{attribute 'GeneratedUsingTerminal: IODEVICETYPE_ETHERCATPROT'}
{attribute addProperty BoxType "IODEVICETYPE_ETHERCATPROT"}
{attribute addProperty Id "DevCtrlAT %Q*UINT2Frm0CtrlAT %Q*UINT2Frm0WcCtrlAT %Q*UINT2Frm1CtrlAT %Q*UINT2Frm1WcCtrlAT %Q*UINT2Frm2CtrlAT %Q*UINT2Frm2WcCtrlAT %Q*UINT2Frm3CtrlAT %Q*UINT2Frm3WcCtrlAT %Q*UINT2Frm4CtrlAT %Q*UINT2Frm4WcCtrlAT %Q*UINT2Frm5CtrlAT %Q*UINT2Frm5WcCtrlAT %Q*UINT2Frm6CtrlAT %Q*UINT2Frm6WcCtrlAT %Q*UINT2Frm7CtrlAT %Q*UINT2Frm7WcCtrlAT %Q*UINT2Frm8CtrlAT %Q*UINT2Frm8WcCtrlAT %Q*UINT2Frm9CtrlAT %Q*UINT2Frm9WcCtrlAT %Q*UINT2Frm10CtrlAT %Q*UINT2Frm10WcCtrlAT %Q*UINT2Frm11CtrlAT %Q*UINT2Frm11WcCtrlAT %Q*UINT2Frm12CtrlAT %Q*UINT2Frm12WcCtrlAT %Q*UINT2Frm13CtrlAT %Q*UINT2Frm13WcCtrlAT %Q*UINT2Frm14CtrlAT %Q*UINT2Frm14WcCtrlAT %Q*UINT2Frm15CtrlAT %Q*UINT2Frm15WcCtrlAT %Q*UINT2Frm16CtrlAT %Q*UINT2Frm16WcCtrlAT %Q*UINT2Frm17CtrlAT %Q*UINT2Frm17WcCtrlAT %Q*UINT2Frm18CtrlAT %Q*UINT2Frm18WcCtrlAT %Q*UINT2Frm19CtrlAT %Q*UINT2Frm19WcCtrlAT %Q*UINT2Frm20CtrlAT %Q*UINT2Frm20WcCtrlAT %Q*UINT2Frm21CtrlAT %Q*UINT2Frm21WcCtrlAT %Q*UINT2Frm22CtrlAT %Q*UINT2Frm22WcCtrlAT %Q*UINT2Frm23CtrlAT %Q*UINT2Frm23WcCtrlAT %Q*UINT2Frm24CtrlAT %Q*UINT2Frm24WcCtrlAT %Q*UINT2Frm25CtrlAT %Q*UINT2Frm25WcCtrlAT %Q*UINT2"}
{attribute addProperty CRC "597139726"}
{attribute addProperty Size "106"}
TYPE Outputs_2397A10E EXTENDS OutputBase_10CEE7DE :
STRUCT
	{attribute addProperty Name "DevCtrl"}
	DevCtrl AT %Q* : UINT;
	{attribute addProperty Name "Frm0Ctrl"}
	Frm0Ctrl AT %Q* : UINT;
	{attribute addProperty Name "Frm0WcCtrl"}
	Frm0WcCtrl AT %Q* : UINT;
	{attribute addProperty Name "Frm1Ctrl"}
	Frm1Ctrl AT %Q* : UINT;
	{attribute addProperty Name "Frm1WcCtrl"}
	Frm1WcCtrl AT %Q* : UINT;
	{attribute addProperty Name "Frm2Ctrl"}
	Frm2Ctrl AT %Q* : UINT;
	{attribute addProperty Name "Frm2WcCtrl"}
	Frm2WcCtrl AT %Q* : UINT;
	{attribute addProperty Name "Frm3Ctrl"}
	Frm3Ctrl AT %Q* : UINT;
	{attribute addProperty Name "Frm3WcCtrl"}
	Frm3WcCtrl AT %Q* : UINT;
	{attribute addProperty Name "Frm4Ctrl"}
	Frm4Ctrl AT %Q* : UINT;
	{attribute addProperty Name "Frm4WcCtrl"}
	Frm4WcCtrl AT %Q* : UINT;
	{attribute addProperty Name "Frm5Ctrl"}
	Frm5Ctrl AT %Q* : UINT;
	{attribute addProperty Name "Frm5WcCtrl"}
	Frm5WcCtrl AT %Q* : UINT;
	{attribute addProperty Name "Frm6Ctrl"}
	Frm6Ctrl AT %Q* : UINT;
	{attribute addProperty Name "Frm6WcCtrl"}
	Frm6WcCtrl AT %Q* : UINT;
	{attribute addProperty Name "Frm7Ctrl"}
	Frm7Ctrl AT %Q* : UINT;
	{attribute addProperty Name "Frm7WcCtrl"}
	Frm7WcCtrl AT %Q* : UINT;
	{attribute addProperty Name "Frm8Ctrl"}
	Frm8Ctrl AT %Q* : UINT;
	{attribute addProperty Name "Frm8WcCtrl"}
	Frm8WcCtrl AT %Q* : UINT;
	{attribute addProperty Name "Frm9Ctrl"}
	Frm9Ctrl AT %Q* : UINT;
	{attribute addProperty Name "Frm9WcCtrl"}
	Frm9WcCtrl AT %Q* : UINT;
	{attribute addProperty Name "Frm10Ctrl"}
	Frm10Ctrl AT %Q* : UINT;
	{attribute addProperty Name "Frm10WcCtrl"}
	Frm10WcCtrl AT %Q* : UINT;
	{attribute addProperty Name "Frm11Ctrl"}
	Frm11Ctrl AT %Q* : UINT;
	{attribute addProperty Name "Frm11WcCtrl"}
	Frm11WcCtrl AT %Q* : UINT;
	{attribute addProperty Name "Frm12Ctrl"}
	Frm12Ctrl AT %Q* : UINT;
	{attribute addProperty Name "Frm12WcCtrl"}
	Frm12WcCtrl AT %Q* : UINT;
	{attribute addProperty Name "Frm13Ctrl"}
	Frm13Ctrl AT %Q* : UINT;
	{attribute addProperty Name "Frm13WcCtrl"}
	Frm13WcCtrl AT %Q* : UINT;
	{attribute addProperty Name "Frm14Ctrl"}
	Frm14Ctrl AT %Q* : UINT;
	{attribute addProperty Name "Frm14WcCtrl"}
	Frm14WcCtrl AT %Q* : UINT;
	{attribute addProperty Name "Frm15Ctrl"}
	Frm15Ctrl AT %Q* : UINT;
	{attribute addProperty Name "Frm15WcCtrl"}
	Frm15WcCtrl AT %Q* : UINT;
	{attribute addProperty Name "Frm16Ctrl"}
	Frm16Ctrl AT %Q* : UINT;
	{attribute addProperty Name "Frm16WcCtrl"}
	Frm16WcCtrl AT %Q* : UINT;
	{attribute addProperty Name "Frm17Ctrl"}
	Frm17Ctrl AT %Q* : UINT;
	{attribute addProperty Name "Frm17WcCtrl"}
	Frm17WcCtrl AT %Q* : UINT;
	{attribute addProperty Name "Frm18Ctrl"}
	Frm18Ctrl AT %Q* : UINT;
	{attribute addProperty Name "Frm18WcCtrl"}
	Frm18WcCtrl AT %Q* : UINT;
	{attribute addProperty Name "Frm19Ctrl"}
	Frm19Ctrl AT %Q* : UINT;
	{attribute addProperty Name "Frm19WcCtrl"}
	Frm19WcCtrl AT %Q* : UINT;
	{attribute addProperty Name "Frm20Ctrl"}
	Frm20Ctrl AT %Q* : UINT;
	{attribute addProperty Name "Frm20WcCtrl"}
	Frm20WcCtrl AT %Q* : UINT;
	{attribute addProperty Name "Frm21Ctrl"}
	Frm21Ctrl AT %Q* : UINT;
	{attribute addProperty Name "Frm21WcCtrl"}
	Frm21WcCtrl AT %Q* : UINT;
	{attribute addProperty Name "Frm22Ctrl"}
	Frm22Ctrl AT %Q* : UINT;
	{attribute addProperty Name "Frm22WcCtrl"}
	Frm22WcCtrl AT %Q* : UINT;
	{attribute addProperty Name "Frm23Ctrl"}
	Frm23Ctrl AT %Q* : UINT;
	{attribute addProperty Name "Frm23WcCtrl"}
	Frm23WcCtrl AT %Q* : UINT;
	{attribute addProperty Name "Frm24Ctrl"}
	Frm24Ctrl AT %Q* : UINT;
	{attribute addProperty Name "Frm24WcCtrl"}
	Frm24WcCtrl AT %Q* : UINT;
	{attribute addProperty Name "Frm25Ctrl"}
	Frm25Ctrl AT %Q* : UINT;
	{attribute addProperty Name "Frm25WcCtrl"}
	Frm25WcCtrl AT %Q* : UINT;
END_STRUCT
END_TYPE

(* stored: Version 1.2.0.0, ProductVersion 3.1.4024.9
   DUT Outputs_2397A10E: Id {a42603a5-821b-465e-b6fb-dacbd987fcb5} *)
